(* IEC 61131-3 sources: Lasal/CPU_5344_V01/Class/ProductsDbV2, 1 file *)

(* ---- ProductsDbV2.st ---- *)
(*!
<Class
	Name               = "ProductsDbV2"
	Revision           = "1.0"
	RealtimeTask       = "false"
	CyclicTask         = "true"
	DefCyclictime      = "10 ms"
	BackgroundTask     = "true"
	DefBackground      = "10 ms"
	Sigmatek           = "false"
	OSInterface        = "false"
	HighPriority       = "false"
	Automatic          = "false"
	UpdateMode         = "Prescan"
	SharedCommandTable = "true"
	Objectsize         = "(600,1500)">
	<Channels>
		<Server Name="endAngle" Visualized="true" Initialize="false" WriteProtected="false" Retentive="false"/>
		<Server Name="frontEndFlipAllowed" Visualized="true" Initialize="false" WriteProtected="false" Retentive="false"/>
		<Server Name="HmiDeleteRecipe" Visualized="true" Initialize="false" WriteProtected="false" Retentive="false"/>
		<Server Name="HmiReloadRecipe" Visualized="true" Initialize="false" WriteProtected="false" Retentive="false"/>
		<Server Name="HmiSaveRecipe" Visualized="true" Initialize="false" WriteProtected="false" Retentive="false"/>
		<Server Name="noEndSaw" Visualized="true" Initialize="false" WriteProtected="false" Retentive="false"/>
		<Server Name="OperationId1" Visualized="true" Initialize="false" WriteProtected="false" Retentive="false"/>
		<Server Name="OperationId2" Visualized="true" Initialize="false" WriteProtected="false" Retentive="false"/>
		<Server Name="OperationId3" Visualized="true" Initialize="false" WriteProtected="false" Retentive="false"/>
		<Server Name="parAutoSave" Visualized="true" Initialize="false" WriteProtected="false" Retentive="File"/>
		<Server Name="ProductHeight" Visualized="true" Initialize="false" WriteProtected="false" Retentive="false"/>
		<Server Name="ProductLength" Visualized="true" Initialize="false" WriteProtected="false" Retentive="false"/>
		<Server Name="ProductWidth" Visualized="true" Initialize="false" WriteProtected="false" Retentive="false"/>
		<Server Name="RecipeId" Visualized="true" Initialize="false" WriteProtected="false" Retentive="SRam"/>
		<Server Name="setZposAtHalfWidth" Visualized="true" Initialize="false" WriteProtected="false" Retentive="SRam"/>
		<Server Name="startAngle" Visualized="true" Initialize="false" WriteProtected="false" Retentive="false"/>
		<Server Name="strDescription" Class="EditString" Visualized="true" Remotely="true" Initialize="true" WriteProtected="false" Retentive="false" Comment="use this channel to access the string functions"/>
		<Server Name="strProductCode" Class="EditString" Visualized="true" Remotely="true" Initialize="true" WriteProtected="false" Retentive="false" Comment="use this channel to access the string functions"/>
		<Server Name="stsUnsafeChanges" Visualized="true" Initialize="false" WriteProtected="true" Retentive="false"/>
		<Server Name="upDownFlipAllowed" Visualized="true" Initialize="false" WriteProtected="false" Retentive="false"/>
		<Client Name="FB" Required="true" Internal="false"/>
		<Client Name="FileSys" Required="false" Internal="false"/>
		<Client Name="OperationData" Required="true" Internal="true"/>
		<Client Name="RamEx" Required="true" Internal="false"/>
		<Client Name="str_Description" Required="true" Internal="true"/>
		<Client Name="str_ProductCode" Required="true" Internal="true"/>
	</Channels>
	<Separators>
		<Servers>
			<SepChn Position="14"/>
			<SepChn Position="16"/>
		</Servers>
		<Clients>
			<SepChn Position="1"/>
		</Clients>
	</Separators>
	<Network Name="ProductsDbV2">
		<!-- List of Components in this network -->
		<Components>
			<Object
				Name       = "_base"
				Class      = "cmBase"
				Position   = "(218,120)"
				Visualized = "true">
				<Channels>
					<Server Name="ClassSvr"/>
					<Server Name="cmdHMI"/>
					<Server Name="ErrorNr"/>
					<Server Name="mode"/>
					<Server Name="state"/>
					<Server Name="stsHMI_RunsAllowed"/>
					<Server Name="stsInAlarm"/>
					<Server Name="stsIsInterlocked"/>
					<Client Name="id"/>
					<Client Name="nwEmOrUnit"/>
				</Channels>
			</Object>
			<Object
				Name       = "OperationData"
				Class      = "OperationDataV2"
				Position   = "(420,1470)"
				Visualized = "true">
				<Channels>
					<Server Name="ClassSvr"/>
					<Server Name="firstIdx"/>
				</Channels>
			</Object>
			<Object
				Name       = "str_Description"
				Class      = "EditString"
				Position   = "(360,810)"
				Visualized = "true"
				Remotely   = "true">
				<Channels>
					<Server Name="Data"/>
					<Server Name="Handle"/>
					<Server Name="NewData"/>
				</Channels>
			</Object>
			<Object
				Name       = "str_ProductCode"
				Class      = "EditString"
				Position   = "(360,1110)"
				Visualized = "true"
				Remotely   = "true">
				<Channels>
					<Server Name="Data"/>
					<Server Name="Handle"/>
					<Server Name="NewData"/>
				</Channels>
			</Object>
		</Components>
		<Comments>
		</Comments>
		<!-- List of Connections in this network -->
		<Connections>
			<Connection Source="this.ClassSvr" Destination="_base.ClassSvr" Vertices="(1058,210),(864,210),"/>
			<Connection Source="this.state" Destination="_base.state" Vertices="(1058,270),(864,270),"/>
			<Connection Source="this.mode" Destination="_base.mode" Vertices="(1058,330),(864,330),"/>
			<Connection Source="this.cmdHMI" Destination="_base.cmdHMI" Vertices="(1058,390),(864,390),"/>
			<Connection Source="this.stsInAlarm" Destination="_base.stsInAlarm" Vertices="(1058,450),(864,510),"/>
			<Connection Source="this.stsIsInterlocked" Destination="_base.stsIsInterlocked" Vertices="(1058,510),(864,570),"/>
			<Connection Source="this.stsHMI_RunsAllowed" Destination="_base.stsHMI_RunsAllowed" Vertices="(1058,570),(864,630),"/>
			<Connection Source="this.ErrorNr" Destination="_base.ErrorNr" Vertices="(1058,630),(864,690),"/>
			<Connection Source="this.str_ProductCode" Destination="str_ProductCode.Data"/>
			<Connection Source="this.str_Description" Destination="str_Description.Data"/>
			<Connection Source="this.OperationData" Destination="OperationData.ClassSvr"/>
			<Connection Source="this.strProductCode" Destination="str_ProductCode.Data" Vertices="(1058,810),(676,1200),"/>
			<Connection Source="this.strDescription" Destination="str_Description.Data" Vertices="(1058,750),(676,900),"/>
			<Connection Source="_base.nwEmOrUnit" Destination="this.nwEmOrUnit" Vertices="(218,210),(38,210),"/>
			<Connection Source="_base.id" Destination="this.id" Vertices="(218,270),(38,270),"/>
		</Connections>
		<!-- Headerfiles -->
		<Options>
		</Options>
	</Network>
</Class>
*)
#pragma using cmBase

ProductsDbV2 : CLASS
: cmBase
	TYPE
	  str_100 : ARRAY [0..225] OF CHAR;
	  str_3000 : ARRAY [0..3000] OF CHAR;
#pragma pack(push, 1)
	  tBewerkingsRegel : STRUCT  //! <Type Public="true" Name="tBewerkingsRegel"/>
	    Bewerking : Units;
	  END_STRUCT;
#pragma pack(pop)
#pragma pack(push, 1)
	  tRecipeLine : STRUCT  //! <Type Public="true" Name="tRecipeLine"/>
	    rnr : DINT;
	    xpos : DINT;
	    ypos : DINT;
	    zpos : DINT;
	    amount : DINT;
	    pitch : DINT;
	    operationId : DINT;
	    operations : Units;
	  END_STRUCT;
#pragma pack(pop)
	  tRecipeLineList : ARRAY [0..cProdDbMaxOperationLines] OF tRecipeLine;  //! <Type Public="true" Name="tRecipeLineList"/>
#pragma pack(push, 1)
	  tRecipeData : STRUCT  //! <Type Public="true" Name="tRecipeData"/>
	    id : DINT;
	    description : gbl_datatypes::tStr20;
	    productCode : gbl_datatypes::tStr20;
	    length : DINT;
	    operationId1 : DINT;
	    operationId2 : DINT;
	    operationId3 : DINT;
	    noEndSaw : DINT;
	    upDownFlipAllowed : DINT;
	    frontEndFilpAllowed : DINT;
	    startAngle : DINT;
	    endAngle : DINT;
	    operations : tRecipeLineList;
	    productWidth : DINT;
	    productHeight : DINT;
	  END_STRUCT;
#pragma pack(pop)
	  tData : ARRAY [0..1] OF tRecipeData;
#pragma pack(push, 1)
	  tOperationtype : STRUCT
	    BU1 : DINT;
	    BU2 : DINT;
	    BU3 : DINT;
	    BU4 : DINT;
	    BU5 : DINT;
	    BU6 : DINT;
	    BU7 : DINT;
	    BU8 : DINT;
	    BU9 : DINT;
	    BU10 : DINT;
	    BU12 : DINT;
	    BU13 : DINT;
	    BU14 : DINT;
	  END_STRUCT;
#pragma pack(pop)
	END_TYPE
  //Servers:
	RecipeId 	: SvrCh_UDINT;
	strDescription 	: SvrChCmd_UDINT;
	strProductCode 	: SvrChCmd_UDINT;
	ProductLength 	: SvrCh_DINT;
	ProductWidth 	: SvrCh_DINT;
	ProductHeight 	: SvrCh_DINT;
	OperationId1 	: SvrCh_DINT;
	OperationId2 	: SvrCh_DINT;
	OperationId3 	: SvrCh_DINT;
	noEndSaw 	: SvrCh_DINT;
	upDownFlipAllowed 	: SvrCh_DINT;
	frontEndFlipAllowed 	: SvrCh_DINT;
	startAngle 	: SvrCh_DINT;
	endAngle 	: SvrCh_DINT;
	setZposAtHalfWidth 	: SvrCh_DINT;
	HmiSaveRecipe 	: SvrCh_DINT;
	HmiReloadRecipe 	: SvrCh_DINT;
	HmiDeleteRecipe 	: SvrCh_DINT;
	stsUnsafeChanges 	: SvrCh_DINT;
	parAutoSave 	: SvrCh_DINT;
  //Clients:
	RamEx 	: CltChCmd_RAMex;
	FileSys 	: CltChCmd__FileSys;
	FB 	: CltChCmd_FileBase;
	str_Description 	: CltChCmd_EditString;
	str_ProductCode 	: CltChCmd_EditString;
	OperationData 	: CltChCmd_OperationDataV2;
  //Variables:
		ActRecipeData 	: tRecipeData;
		tempRecipe 	: tRecipeData;
		sizeRecipedata 	: UDINT;
		emptyRecipe 	: tRecipeData;
		tmpText 	: tekst;
		dbAmountOfRecipes 	: UDINT;
		dbAmountOfLinesInRecipe 	: UDINT;
		checkForStorageProductData 	: tRecipeData;
		tmrAutoSave 	: UDINT;
		tmpNrDelete 	: UDINT;
		tmpInputNr 	: UDINT;
		stsRamResult 	: UINT;
  //Functions:

	FUNCTION VIRTUAL GLOBAL Background
		VAR_INPUT
			EAX 	: UDINT;
		END_VAR
		VAR_OUTPUT
			state (EAX) 	: UDINT;
		END_VAR;

	FUNCTION VIRTUAL Init1;

	FUNCTION GLOBAL GetRecipe
		VAR_INPUT
			id 	: DINT;
		END_VAR
		VAR_OUTPUT
			oRecipe 	: tRecipeData;
		END_VAR;

	FUNCTION UpdateServers;

	FUNCTION GLOBAL giveText
		VAR_INPUT
			progNr 	: DINT;
		END_VAR
		VAR_OUTPUT
			text 	: tekst;
		END_VAR;

	FUNCTION saveRecipe
		VAR_INPUT
			nr 	: UDINT;
			recipe 	: tRecipeData;
		END_VAR
		VAR_OUTPUT
			ok 	: DINT;
		END_VAR;

	FUNCTION loadRecipe
		VAR_INPUT
			nr 	: UDINT;
		END_VAR
		VAR_OUTPUT
			ok 	: DINT;
		END_VAR;

	FUNCTION saveChanges
		VAR_OUTPUT
			ok 	: DINT;
		END_VAR;

	FUNCTION VIRTUAL GLOBAL RecipeId::Write
		VAR_INPUT
			input (EAX) 	: UDINT;
		END_VAR
		VAR_OUTPUT
			result (EAX) 	: UDINT;
		END_VAR;

	FUNCTION VIRTUAL GLOBAL strDescription::Read
		VAR_OUTPUT
			output (EAX) 	: UDINT;
		END_VAR;

	FUNCTION VIRTUAL GLOBAL strDescription::Write
		VAR_INPUT
			input (EAX) 	: UDINT;
		END_VAR
		VAR_OUTPUT
			result (EAX) 	: UDINT;
		END_VAR;

	FUNCTION VIRTUAL GLOBAL strProductCode::Read
		VAR_OUTPUT
			output (EAX) 	: UDINT;
		END_VAR;

	FUNCTION VIRTUAL GLOBAL strProductCode::Write
		VAR_INPUT
			input (EAX) 	: UDINT;
		END_VAR
		VAR_OUTPUT
			result (EAX) 	: UDINT;
		END_VAR;

	FUNCTION VIRTUAL GLOBAL ProductLength::Write
		VAR_INPUT
			input (EAX) 	: DINT;
		END_VAR
		VAR_OUTPUT
			result (EAX) 	: DINT;
		END_VAR;

	FUNCTION VIRTUAL GLOBAL ProductWidth::Write
		VAR_INPUT
			input (EAX) 	: DINT;
		END_VAR
		VAR_OUTPUT
			result (EAX) 	: DINT;
		END_VAR;

	FUNCTION VIRTUAL GLOBAL ProductHeight::Write
		VAR_INPUT
			input (EAX) 	: DINT;
		END_VAR
		VAR_OUTPUT
			result (EAX) 	: DINT;
		END_VAR;

	FUNCTION VIRTUAL GLOBAL OperationId1::Write
		VAR_INPUT
			input (EAX) 	: DINT;
		END_VAR
		VAR_OUTPUT
			result (EAX) 	: DINT;
		END_VAR;

	FUNCTION VIRTUAL GLOBAL OperationId2::Write
		VAR_INPUT
			input (EAX) 	: DINT;
		END_VAR
		VAR_OUTPUT
			result (EAX) 	: DINT;
		END_VAR;

	FUNCTION VIRTUAL GLOBAL OperationId3::Write
		VAR_INPUT
			input (EAX) 	: DINT;
		END_VAR
		VAR_OUTPUT
			result (EAX) 	: DINT;
		END_VAR;

	FUNCTION VIRTUAL GLOBAL noEndSaw::Write
		VAR_INPUT
			input (EAX) 	: DINT;
		END_VAR
		VAR_OUTPUT
			result (EAX) 	: DINT;
		END_VAR;

	FUNCTION VIRTUAL GLOBAL upDownFlipAllowed::Write
		VAR_INPUT
			input (EAX) 	: DINT;
		END_VAR
		VAR_OUTPUT
			result (EAX) 	: DINT;
		END_VAR;

	FUNCTION VIRTUAL GLOBAL frontEndFlipAllowed::Write
		VAR_INPUT
			input (EAX) 	: DINT;
		END_VAR
		VAR_OUTPUT
			result (EAX) 	: DINT;
		END_VAR;

	FUNCTION VIRTUAL GLOBAL startAngle::Write
		VAR_INPUT
			input (EAX) 	: DINT;
		END_VAR
		VAR_OUTPUT
			result (EAX) 	: DINT;
		END_VAR;

	FUNCTION VIRTUAL GLOBAL endAngle::Write
		VAR_INPUT
			input (EAX) 	: DINT;
		END_VAR
		VAR_OUTPUT
			result (EAX) 	: DINT;
		END_VAR;

	FUNCTION VIRTUAL GLOBAL HmiSaveRecipe::Write
		VAR_INPUT
			input (EAX) 	: DINT;
		END_VAR
		VAR_OUTPUT
			result (EAX) 	: DINT;
		END_VAR;

	FUNCTION VIRTUAL GLOBAL HmiReloadRecipe::Write
		VAR_INPUT
			input (EAX) 	: DINT;
		END_VAR
		VAR_OUTPUT
			result (EAX) 	: DINT;
		END_VAR;

	FUNCTION VIRTUAL GLOBAL HmiDeleteRecipe::Write
		VAR_INPUT
			input (EAX) 	: DINT;
		END_VAR
		VAR_OUTPUT
			result (EAX) 	: DINT;
		END_VAR;

	FUNCTION VIRTUAL GLOBAL stsUnsafeChanges::Read
		VAR_OUTPUT
			output (EAX) 	: DINT;
		END_VAR;
  //Tables:
	FUNCTION @STD
		VAR_OUTPUT
			ret_code	: CONFSTATES;
		END_VAR;
	FUNCTION GLOBAL TAB @CT_;
END_CLASS;

#pragma using EditString
#pragma using OperationDataV2
#pragma usingLtd _FileSys
#pragma usingLtd FileBase
#pragma usingLtd RAMex

// JdK 29-11-2019 productsDBV2 created to handle 'recipes' like products, assembly's etc.
// functions like autosave, save, save as, reload (undo changes) are available
// storage to usb and load from usb are not yet functional, will be added later

//
//ErrorNr 1 no file present
//ErrorNr 2 USB not present
//ErrorNr 3 cannot open file
//ErrorNr 4 error reading file
//ErrorNr 5 wrong format
//ErrorNr 6 too many lines
//ErrorNr 7 too little chars in data string

FUNCTION VIRTUAL ProductsDbV2::Init1

  IF initDone= 0 THEN

    dbAmountOfRecipes:= CPRODDBMAXPRODUCTS; //read in amounts
    dbAmountOfLinesInRecipe:= CPRODDBMAXOPERATIONLINES;
    sizeRecipedata := to_udint(sizeof(tRecipeData)); //put size of product data in var
    _memset(dest:=#emptyRecipe, usByte:=0, cntr:=sizeRecipedata); //set empty product

    IF RamEx.GetSize() <> (sizeRecipedata*dbAmountOfRecipes) THEN //check if ram size isn't set yet
      IF RamEx.SetSize(udsize:= (sizeRecipedata*dbAmountOfRecipes)) = C_OK THEN //only if setting is done, say init is done
        initDone:= 1;

        loadRecipe(nr:=RecipeId); //after setting size of db try to load the recipe

      END_IF;
    ELSE
      initDone:= 1;
      loadRecipe(nr:=RecipeId); //also if size is ok, load recipe
    END_IF;

  END_IF;

END_FUNCTION

FUNCTION VIRTUAL GLOBAL ProductsDbV2::Background
	VAR_INPUT
		EAX 	: UDINT;
	END_VAR
	VAR_OUTPUT
		state (EAX) 	: UDINT;
	END_VAR

  //check if we need to update the strings
  if str_Description.NewData.Read() <> 0 then//description
    _memset(dest:=#ActRecipeData.description[0], usByte:=0, cntr:=sizeof(ActRecipeData.description));
    str_Description.ReadDataOff(udOff:=0, pData:=#ActRecipeData.description[0], udMax:=sizeof(ActRecipeData.description));
    str_Description.NewData.Write(input:=0);
  end_if;

  if str_ProductCode.NewData.Read() <> 0 then//productCode
    _memset(dest:=#ActRecipeData.productCode[0], usByte:=0, cntr:=sizeof(ActRecipeData.productCode));
    str_ProductCode.ReadDataOff(udOff:=0, pData:=#ActRecipeData.productCode[0], udMax:=sizeof(ActRecipeData.productCode));
    str_ProductCode.NewData.Write(input:=0);
  end_if;

  //if autosave is active, check every ten seconds if we should save
  IF parAutoSave & ops.tAbsolute-tmrAutoSave> 10000 THEN
    saveChanges();
    tmrAutoSave:= ops.tAbsolute;
  END_IF;

  IF HmiDeleteRecipe= -10 THEN //means delete complete db
    IF tmpNrDelete > 0 & tmpNrDelete < dbAmountOfRecipes THEN
      IF saveRecipe(nr:=tmpNrDelete, recipe:=emptyRecipe)= 1 THEN
        tmpNrDelete+=1;
        IF tmpNrDelete = dbAmountOfRecipes THEN
          HmiDeleteRecipe:= 0; //all recipes are deleted now
          loadRecipe(nr:=RecipeId);//load active recipe to show it's empty
        END_IF;
      END_IF;
    END_IF;
  END_IF;

  stsUnsafeChanges.Read();

  state:= 0;

END_FUNCTION

FUNCTION VIRTUAL GLOBAL ProductsDbV2::stsUnsafeChanges::Read
	VAR_OUTPUT
		output (EAX) 	: DINT;
	END_VAR

  IF ActRecipeData <> checkForStorageProductData THEN
    stsUnsafeChanges:= 1;
  ELSE
    stsUnsafeChanges:= 0;
  END_IF;

	output := stsUnsafeChanges;

END_FUNCTION

FUNCTION VIRTUAL GLOBAL ProductsDbV2::RecipeId::Write
	VAR_INPUT
		input (EAX) 	: UDINT;
	END_VAR
	VAR_OUTPUT
		result (EAX) 	: UDINT;
	END_VAR

  IF input > 0 & input < dbAmountOfRecipes THEN //we don't use nr 0, so we have one less
    IF parAutoSave= 0 | saveChanges()= 1 THEN //only if autosave is active, else in screen project choose to save or not should be made before writing a new product ID
      RecipeId:= input; //keep input in memory
      loadRecipe(nr:=RecipeId);
    END_IF;

  ELSE
    Result := Access_Denied;
  End_If;

END_FUNCTION

FUNCTION ProductsDbV2::saveRecipe
	VAR_INPUT
		nr 	: UDINT;
		recipe 	: tRecipeData;
	END_VAR
	VAR_OUTPUT
		ok 	: DINT;
	END_VAR

  //function save recipe in input nr in ram db
  IF nr > 0 & nr < dbAmountOfRecipes THEN //we don't use nr 0, so we have one less
    tempRecipe:= recipe;
    stsRamResult:= RamEx.SetDataAt(pdata:=#tempRecipe$usint, udsize:=sizeRecipedata, udat:=nr * sizeRecipedata);
    IF stsRamResult= 5 THEN
      ok:= 1;
    ELSE
      ok:= 0;
    END_IF;
  ELSE
    ok:= 0;
  END_IF;

END_FUNCTION

FUNCTION ProductsDbV2::loadRecipe
	VAR_INPUT
		nr 	: UDINT;
	END_VAR
	VAR_OUTPUT
		ok 	: DINT;
	END_VAR

  //function loads recipe from nr into act recipe, also changes check saving recipe, used to control if saving is required
  IF nr>0 & nr<dbAmountOfRecipes THEN
    stsRamResult:= RamEx.GetDataAt(pData:=#ActRecipeData$USINT, udSize:=sizeRecipedata, udAt:=nr* sizeRecipedata);
    IF stsRamResult= 5 THEN
      checkForStorageProductData:= ActRecipeData; //no changes yet
      UpdateServers();
      ok:= 1;
    ELSE
      ok:= 0;
    END_IF;
  ELSE
    ok:= 0;
  END_IF;

END_FUNCTION

FUNCTION ProductsDbV2::saveChanges
	VAR_OUTPUT
		ok 	: DINT;
	END_VAR

  IF checkForStorageProductData <> ActRecipeData THEN //only do saving if there is a difference
    IF saveRecipe(nr:=RecipeId, recipe:=ActRecipeData) THEN
      checkForStorageProductData:= ActRecipeData;
      ok:= 1;
    ELSE
      ok:= 0;
    END_IF;
  ELSE
    ok:= 1; //no changes, means no storage needed
  END_IF;

END_FUNCTION

FUNCTION ProductsDbV2::UpdateServers

//put data of new recipe into data servers
  ProductLength := ActRecipeData.length;
  operationId1 := ActRecipeData.operationId1;
  OperationId2 := ActRecipeData.OperationId2;
  OperationId3 := ActRecipeData.OperationId3;
  noEndSaw     := ActRecipeData.noEndSaw;
  ProductWidth := ActRecipeData.productWidth;
  ProductHeight := ActRecipeData.productHeight;
  upDownFlipAllowed := ActRecipeData.upDownFlipAllowed;
  frontEndFlipAllowed := ActRecipeData.frontEndFilpAllowed;
  //tp 22-04-2020 set angles to 90 if is zero
  if ActRecipeData.startAngle = 0 then
    ActRecipeData.startAngle:=900;
  end_if;
  startAngle := ActRecipeData.startAngle;
  if ActRecipeData.endAngle = 0 then
    ActRecipeData.endAngle:=900;
  end_if;
  endAngle := ActRecipeData.endAngle;

  OperationData.WritePtrs(ptr:=#ActRecipeData.operations, ptrProdHeigth:=#ActRecipeData.productHeight, useHeigth:=setZposAtHalfWidth, maxLines:=to_dint(dbAmountOfLinesInRecipe));
  str_Description.WriteDataOff(udLen:=sizeof(ActRecipeData.description), udOff:=0, pData:=#ActRecipeData.description[0]);
  str_ProductCode.WriteDataOff(udLen:=sizeof(ActRecipeData.productCode), udOff:=0, pData:=#ActRecipeData.productCode[0]);

END_FUNCTION

////////////////////////////////////////////////////////////////////
// some functions for controlling recipe from HMI

FUNCTION VIRTUAL GLOBAL ProductsDbV2::HmiSaveRecipe::Write
	VAR_INPUT
		input (EAX) 	: DINT;
	END_VAR
	VAR_OUTPUT
		result (EAX) 	: DINT;
	END_VAR

  //function to save actual recipe into given nr
  //if used as regular save, write product id into this server to save,
  //else write nr. where you want to save it
  tmpInputNr:=to_udint(input);
  IF input> 0 & tmpInputNr < dbAmountOfRecipes THEN
    IF saveRecipe(nr:=tmpInputNr, recipe:=ActRecipeData) = 1 THEN
	    HmiSaveRecipe := 0; //saving done
    ELSE
      HmiSaveRecipe:= -1;
    END_IF;
  ELSE
    HmiSaveRecipe := -1; //saving not ok
  END_IF;
	result := HmiSaveRecipe;

END_FUNCTION

FUNCTION VIRTUAL GLOBAL ProductsDbV2::HmiReloadRecipe::Write
	VAR_INPUT
		input (EAX) 	: DINT;
	END_VAR
	VAR_OUTPUT
		result (EAX) 	: DINT;
	END_VAR

  //means throw away all made changes
  IF loadRecipe(nr:=RecipeId)= 1 THEN
  	HmiReloadRecipe := 0; //done
  ELSE
    HmiReloadRecipe := -1; //not ok
  END_IF;

	result := HmiReloadRecipe;

END_FUNCTION

FUNCTION VIRTUAL GLOBAL ProductsDbV2::HmiDeleteRecipe::Write
	VAR_INPUT
		input (EAX) 	: DINT;
	END_VAR
	VAR_OUTPUT
		result (EAX) 	: DINT;
	END_VAR

  //delete all recipes (if value = -10), or one (if value is between min and max recipes)
  tmpInputNr:=to_udint(input);
  IF input = -10 THEN
    HmiDeleteRecipe := input;
    tmpNrDelete:= 1;
  ELSIF input>0 & tmpInputNr < dbAmountOfRecipes THEN
    IF saveRecipe(nr:=tmpInputNr, recipe:=emptyRecipe) = 1 THEN
      IF tmpInputNr = RecipeId THEN //if actual recipe is deleted, reload it
        loadRecipe(nr:=RecipeId);
      END_IF;
      HmiDeleteRecipe:= 0;
    ELSE
      HmiDeleteRecipe:= -1;
    END_IF;
  END_IF;
	result := HmiDeleteRecipe;

END_FUNCTION

/////////////////////////////////////////////////////////////////
// USB functions
//////////////////////////////////////////////////////////////////
// function to get prog from other class

FUNCTION GLOBAL ProductsDbV2::GetRecipe
	VAR_INPUT
		id 	: DINT;
	END_VAR
	VAR_OUTPUT
		oRecipe 	: tRecipeData;
	END_VAR

  if id >= 0 & id < to_dint(dbAmountOfRecipes) then
    if id = to_dint(RecipeId) then //JdK if product is active, just give it back, else db isn't written in right way
      tempRecipe:=ActRecipeData;
    else
      RamEx.GetDataAt(pdata:=#tempRecipe$usint, udsize:=sizeRecipedata, udat:= to_udint(id) * sizeRecipedata);
    end_if;
    oRecipe := tempRecipe;
  else
    oRecipe := emptyRecipe;
  end_if;

END_FUNCTION

//////////////////////////////////////////////////////////////
// functions to write data

FUNCTION VIRTUAL GLOBAL ProductsDbV2::strDescription::Read
	VAR_OUTPUT
		output (EAX) 	: UDINT;
	END_VAR

	strDescription := str_Description.Data.Read();
	output := strDescription;

END_FUNCTION

FUNCTION VIRTUAL GLOBAL ProductsDbV2::strDescription::Write
	VAR_INPUT
		input (EAX) 	: UDINT;
	END_VAR
	VAR_OUTPUT
		result (EAX) 	: UDINT;
	END_VAR

	strDescription := input;
	result := (str_Description.Data.Write(strDescription))$UDINT;
  _memset(dest:=#ActRecipeData.description[0], usByte:=0, cntr:=sizeof(ActRecipeData.description));
  str_Description.ReadDataOff(udOff:=0, pData:=#ActRecipeData.description[0], udMax:=sizeof(ActRecipeData.description));

END_FUNCTION

FUNCTION VIRTUAL GLOBAL ProductsDbV2::strProductCode::Read
	VAR_OUTPUT
		output (EAX) 	: UDINT;
	END_VAR

	strProductCode := str_ProductCode.Data.Read();
	output := strProductCode;

END_FUNCTION

FUNCTION VIRTUAL GLOBAL ProductsDbV2::strProductCode::Write
	VAR_INPUT
		input (EAX) 	: UDINT;
	END_VAR
	VAR_OUTPUT
		result (EAX) 	: UDINT;
	END_VAR

	strProductCode := input;
	result := (str_ProductCode.Data.Write(strProductCode))$UDINT;

END_FUNCTION

FUNCTION VIRTUAL GLOBAL ProductsDbV2::ProductLength::Write
	VAR_INPUT
		input (EAX) 	: DINT;
	END_VAR
	VAR_OUTPUT
		result (EAX) 	: DINT;
	END_VAR

	ProductLength := input;
  ActRecipeData.length := ProductLength;
	result := ProductLength;

END_FUNCTION

FUNCTION VIRTUAL GLOBAL ProductsDbV2::OperationId1::Write
	VAR_INPUT
		input (EAX) 	: DINT;
	END_VAR
	VAR_OUTPUT
		result (EAX) 	: DINT;
	END_VAR

	operationId1 := input;
  ActRecipeData.operationId1 := operationId1;
	result := operationId1;

END_FUNCTION

FUNCTION VIRTUAL GLOBAL ProductsDbV2::OperationId2::Write
	VAR_INPUT
		input (EAX) 	: DINT;
	END_VAR
	VAR_OUTPUT
		result (EAX) 	: DINT;
	END_VAR

	OperationId2 := input;
  ActRecipeData.OperationId2 := OperationId2;
	result := OperationId2;

END_FUNCTION

FUNCTION VIRTUAL GLOBAL ProductsDbV2::OperationId3::Write
	VAR_INPUT
		input (EAX) 	: DINT;
	END_VAR
	VAR_OUTPUT
		result (EAX) 	: DINT;
	END_VAR

	OperationId3 := input;
  ActRecipeData.OperationId3 := OperationId3;
	result := OperationId3;

END_FUNCTION

FUNCTION VIRTUAL GLOBAL ProductsDbV2::ProductWidth::Write
	VAR_INPUT
		input (EAX) 	: DINT;
	END_VAR
	VAR_OUTPUT
		result (EAX) 	: DINT;
	END_VAR

	ProductWidth := input;
  ActRecipeData.productWidth := ProductWidth;
	result := ProductWidth;

END_FUNCTION

FUNCTION VIRTUAL GLOBAL ProductsDbV2::ProductHeight::Write
	VAR_INPUT
		input (EAX) 	: DINT;
	END_VAR
	VAR_OUTPUT
		result (EAX) 	: DINT;
	END_VAR

	ProductHeight := input;
  ActRecipeData.productHeight := ProductHeight;
	result := ProductHeight;

END_FUNCTION

FUNCTION VIRTUAL GLOBAL ProductsDbV2::upDownFlipAllowed::Write
	VAR_INPUT
		input (EAX) 	: DINT;
	END_VAR
	VAR_OUTPUT
		result (EAX) 	: DINT;
	END_VAR

	upDownFlipAllowed := input;
  ActRecipeData.upDownFlipAllowed:= upDownFlipAllowed;
	result := upDownFlipAllowed;

END_FUNCTION

FUNCTION VIRTUAL GLOBAL ProductsDbV2::frontEndFlipAllowed::Write
	VAR_INPUT
		input (EAX) 	: DINT;
	END_VAR
	VAR_OUTPUT
		result (EAX) 	: DINT;
	END_VAR

	frontEndFlipAllowed := input;
  ActRecipeData.frontEndFilpAllowed:= frontEndFlipAllowed;
	result := frontEndFlipAllowed;

END_FUNCTION

FUNCTION VIRTUAL GLOBAL ProductsDbV2::startAngle::Write
	VAR_INPUT
		input (EAX) 	: DINT;
	END_VAR
	VAR_OUTPUT
		result (EAX) 	: DINT;
	END_VAR

  IF input > 0 & input < 1800 THEN
	  startAngle := input;
    ActRecipeData.startAngle:=startAngle;
  END_IF;
	result := startAngle;

END_FUNCTION

FUNCTION VIRTUAL GLOBAL ProductsDbV2::endAngle::Write
	VAR_INPUT
		input (EAX) 	: DINT;
	END_VAR
	VAR_OUTPUT
		result (EAX) 	: DINT;
	END_VAR

  IF input > 0 & input < 1800 THEN
  	endAngle := input;
    ActRecipeData.endAngle:=endAngle;
  END_IF;
	result := endAngle;

END_FUNCTION

FUNCTION VIRTUAL GLOBAL ProductsDbV2::noEndSaw::Write
	VAR_INPUT
		input (EAX) 	: DINT;
	END_VAR
	VAR_OUTPUT
		result (EAX) 	: DINT;
	END_VAR

  IF input >= 0 & input <= 1 THEN
	  noEndSaw := input;
    ActRecipeData.noEndSaw:= noEndSaw;
  END_IF;
	result := noEndSaw;

END_FUNCTION

FUNCTION GLOBAL ProductsDbV2::giveText
	VAR_INPUT
		progNr 	: DINT;
	END_VAR
	VAR_OUTPUT
		text 	: tekst;
	END_VAR

  _memset(dest:=#tmpText[0], usByte:=0, cntr:=sizeof(tmpText));

  if progNr >= 0 & progNr < cProdDbMaxProducts then
    if progNr = to_dint(RecipeId) then //JdK if product is active, just give it back, else db isn't written in right way
      tempRecipe:=ActRecipeData;
    else
      RamEx.GetDataAt(pdata:=#tempRecipe$usint, udsize:=sizeof(tRecipeData), udat:= to_udint(id) * sizeof(tRecipeData));
    end_if;
    _memcpy(ptr1:=#tmpText[0], ptr2:=#tempRecipe.description[0], cntr:=21); //copy all 21 chars to tmp

  end_if;

  text:= tmpText;

END_FUNCTION
